(* LS Electric XG5000 project: traffic_PLC *)
(* PLC LSPLC *)

PROGRAM NewProgram (* task: 스캔 프로그램 *)
VAR
    보행버튼 AT %IX0.0.0 : BOOL;
    보행자녹색 AT %QX0.1.3 : BOOL;
    보행자녹색10초 : TON;
    보행자녹색1초 : TON;
    보행자녹색1초2 : TON;
    보행자적색 AT %QX0.1.4 : BOOL;
    자가유지 AT %MX0 : BOOL;
    차선녹색 AT %QX0.1.0 : BOOL;
    차선녹색타이머 : TON;
    차선적색 AT %QX0.1.2 : BOOL;
    차선적색타이머 : TON;
    차선황색 AT %QX0.1.1 : BOOL;
    차선황색타이머 : TON;
END_VAR

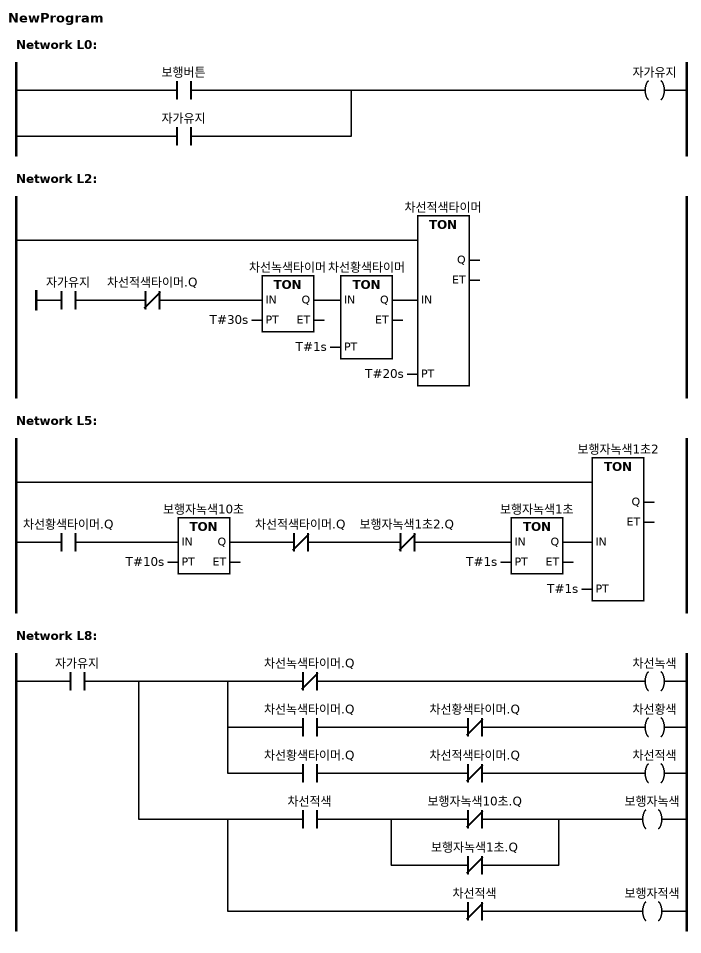
(* Rung L0 *)
자가유지 := 보행버튼 OR 자가유지;
(* Rung L2 *)
차선녹색타이머(IN := 자가유지 AND NOT 차선적색타이머.Q, PT := T#30s);
차선황색타이머(IN := 차선녹색타이머.Q, PT := T#1s);
차선적색타이머(IN := 차선황색타이머.Q, PT := T#20s);
(* Rung L5 *)
보행자녹색10초(IN := 차선황색타이머.Q, PT := T#10s);
보행자녹색1초(IN := 보행자녹색10초.Q AND NOT 차선적색타이머.Q AND NOT 보행자녹색1초2.Q, PT := T#1s);
보행자녹색1초2(IN := 보행자녹색1초.Q, PT := T#1s);
(* Rung L8 *)
차선녹색 := 자가유지 AND NOT 차선녹색타이머.Q;
차선황색 := 자가유지 AND 차선녹색타이머.Q AND NOT 차선황색타이머.Q;
차선적색 := 자가유지 AND 차선황색타이머.Q AND NOT 차선적색타이머.Q;
보행자녹색 := 자가유지 AND 차선적색 AND (NOT 보행자녹색10초.Q OR NOT 보행자녹색1초.Q);
보행자적색 := 자가유지 AND NOT 차선적색;
END_PROGRAM